FUNCTION_BLOCK ClamperSnapSide EXTENDS RunUnitSlave
VAR_INPUT
END_VAR
VAR_OUTPUT
END_VAR
VAR
END_VAR

END_FUNCTION_BLOCK

(* stored: Version 1.1.0.1, ProductVersion 3.1.4024.0
   POU ClamperSnapSide: Id {c14fe538-a423-480e-b144-3ced6a766222}, SpecialFunc None *)
